FUNCTION rt_atan2d : LREAL
VAR_INPUT
	u0: LREAL;
	u1: LREAL;
END_VAR
VAR
END_VAR



IF u1 > 0.0 THEN 
    rt_atan2d := ATAN(u0 / u1);
ELSIF u1 < 0.0 THEN 

    IF u0 >= 0.0 THEN 
        rt_atan2d := 1.0;
    ELSE 
        rt_atan2d := -1.0;
    END_IF;

    rt_atan2d := ATAN(u0 / u1) + (rt_atan2d * 3.1415926535897931);
ELSE 

    IF u0 < 0.0 THEN 
        rt_atan2d := -1.0;
    ELSIF u0 > 0.0 THEN 
        rt_atan2d := 1.0;
    ELSE 
        rt_atan2d := u0;
    END_IF;

    rt_atan2d := rt_atan2d * 1.5707963267948966;
END_IF;

END_FUNCTION

(* stored: Version 1.1.0.1, ProductVersion 3.1.4022.7
   POU rt_atan2d: Id {beed4355-8fba-4ef2-acfb-f6fd6d5fd363}, SpecialFunc None *)
